TYPE ELL14kAttenuationFilterConfig EXTENDS DeviceConfiguration :
STRUCT
	SerialCommunication : SerialCommunication;
END_STRUCT
END_TYPE

(* stored: Version 1.1.0.1, ProductVersion 3.1.4024.4
   DUT ELL14kAttenuationFilterConfig: Id {41021eb4-41cd-4a35-a8b2-2027f10fa406} *)
